RoboDK station: fairino_dk_02.rdk

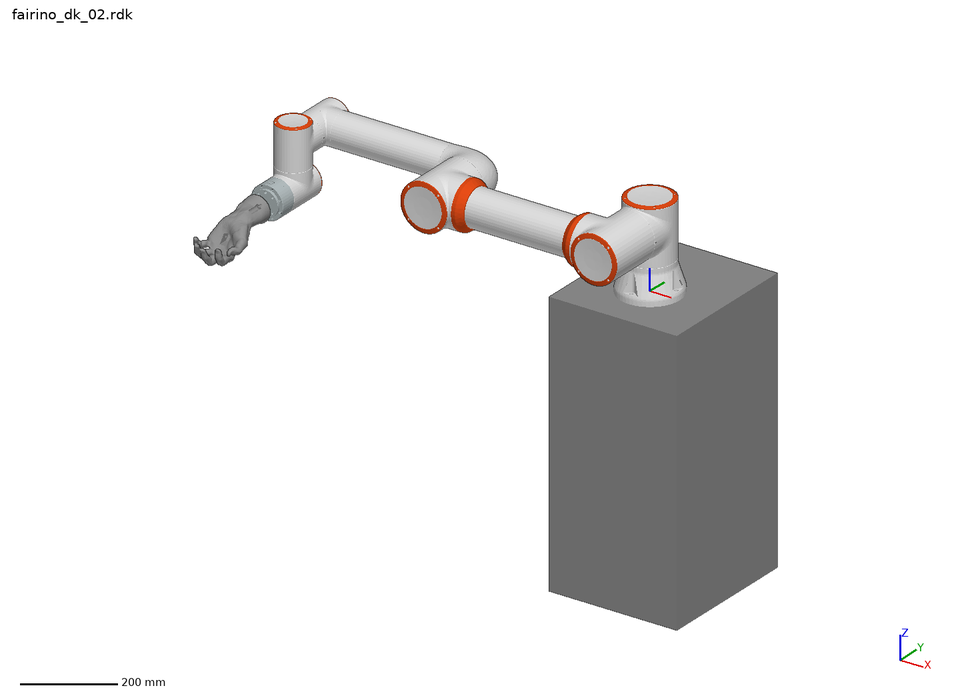
[picture v0: the station drawn from its stored meshes, robots at their saved joint values, targets as dots, program paths as lines]
Station fairino_dk_02 (saved by RoboDK 6.0.4). Poses are relative to the parent item; angles as X-Y-Z fixed-axis rotations.
  - frame Frame 1 at (0, 1000, 0) mm
    - robot FAIRINO FR3 WML input (model FAIRINO FR5): 6 axes
        modified DH rows (alpha deg, a mm, theta deg, d mm): 0, 0, 0, 152; 90, 0, 180, 0; 0, 425, 0, 0; 0, 395, 0, 102; -90, 0, 0, 102; 90, 0, 180, 100
        joint limits [-175, -265, -160, -265, -175, -355] to [175, 85, 160, 85, 175, 355]; home [0, -90, -90, 0, 90, 0]; saved at [0, 0, 0, 0, 0, 0]
      - tool hand_ballholding_noodlev5, TCP at (0, 0, 0) mm, size 105.6 x 194.6 x 100.7 mm, geometry from hand_ballholding_noodlev5.stl
    - object case collision model at (0, 0, 0) mm, size 360 x 320 x 670 mm, geometry from case collision model.stl
  - Python program OSC_receive_pos (listed below)

--- Python program OSC_receive_pos ---
from robodk import robolink
from pythonosc import udp_client
from pythonosc.osc_server import BlockingOSCUDPServer
from pythonosc.dispatcher import Dispatcher

# --- Configuration ---
ROBOT_NAME = 'FAIRINO FR3 WML input'
OSC_IN_IP = "127.0.0.1"
OSC_IN_PORT = 8100

# Initialize RoboDK
RDK = robolink.Robolink()
robot = RDK.Item(ROBOT_NAME, robolink.ITEM_TYPE_ROBOT)

def handle_joints(address, *args):
    joints = [float(a) for a in args]
    robot.setJoints(joints)

# --- OSC Server Setup ---
dispatcher = Dispatcher()
dispatcher.map("/joints", handle_joints)

print(f"Listening on {OSC_IN_IP}:{OSC_IN_PORT}")
print(f"Mirroring joints to '{ROBOT_NAME}'...")

server = BlockingOSCUDPServer((OSC_IN_IP, OSC_IN_PORT), dispatcher)
server.serve_forever()
